SUBAPPLICATION Button_IXA_TO_Remote_WRITE_BG_OPC (* VT-Button lesen + Remote-OPC-UA-Write an Zielmodul + VT-Hintergrundfarbe aus Remote-Subscribe (generisch, ein Kanal, fuer Ausgaenge auf Modulen ohne eigene VT-Anbindung) *)
  (* Standard: 61499-2 *)
  (* Version 1.0, 2026-08-27, franz, Meisterschulen am Ostbahnhof *)
  PACKAGE MyLib::sys;
  IMPORT isobus::UT::Q::const::IDs::ID_NULL;
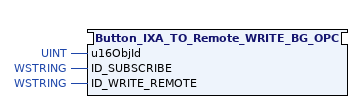
  VAR_INPUT
    u16ObjId : UINT := ID_NULL; (* Object ID Button/Hintergrund (VT) *)
    ID_SUBSCRIBE : WSTRING; (* Remote-Subscribe-Adresse (Status/Farbe, ACTION=SUBSCRIBE) *)
    ID_WRITE_REMOTE : WSTRING; (* Remote-Write-Adresse zum Zielmodul (Befehl, ACTION=WRITE, CLIENT) *)
  END_VAR
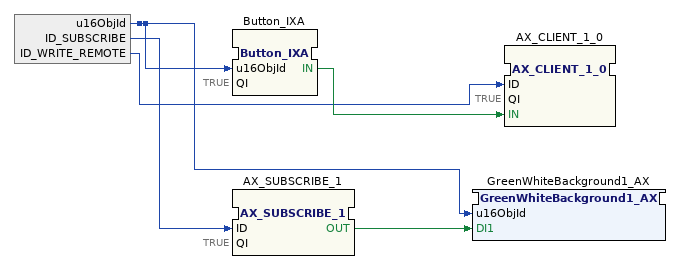
  FBS
    Button_IXA : isobus::UT::io::Button::Button_IXA(QI := TRUE);
    AX_CLIENT_1_0 : adapter::net::AX_CLIENT_1_0(QI := TRUE);
    AX_SUBSCRIBE_1 : adapter::net::AX_SUBSCRIBE_1(QI := TRUE);
  END_FBS
  SUBAPPS
    GreenWhiteBackground1_AX : MyLib::sys::GreenWhiteBackground1_AX;
  END_SUBAPPS
  DATA_CONNECTIONS
    u16ObjId TO Button_IXA.u16ObjId;
    u16ObjId TO GreenWhiteBackground1_AX.u16ObjId;
    ID_SUBSCRIBE TO AX_SUBSCRIBE_1.ID;
    ID_WRITE_REMOTE TO AX_CLIENT_1_0.ID;
  END_CONNECTIONS
  ADAPTER_CONNECTIONS
    Button_IXA.IN TO AX_CLIENT_1_0.IN;
    AX_SUBSCRIBE_1.OUT TO GreenWhiteBackground1_AX.DI1;
  END_CONNECTIONS
END_SUBAPPLICATION
